TYPE STMControl :
STRUCT
	enable : BOOL;
	reset : BOOL;
	invertDirection : BOOL;
	brakeOutput : BOOL;
END_STRUCT
END_TYPE

(* stored: Version 1.1.0.1, ProductVersion 3.1.4024.9
   DUT STMControl: Id {2c1a434e-43a8-47b9-a1e1-cba6905cd6b9} *)
